# B&R Automation Studio project mappViewGettingStarted
Automation Studio 4.3.3.196; technology packages: mappView 1.3.0

## Configuration Config1

CPU PC_any, AutomationRuntime I4.33, Build 4.1.2, Vc V4.25.0

### Hardware
```
PC : PC_any v1.1.0.0 (OrderNumber=PC)
  ConfigurationID = mappViewGettingStarted_Config1
  ActivateOpcUa = 1
```

## Logical view

### Program Logical/Program (IEC)

#### Variables.var
```iecst
VAR
	MTBasicsPT1_0 : MTBasicsPT1;
	aiTankLevel : USINT;
	arrayVm : ARRAY[0..99] OF UINT;
	i : INT;
END_VAR
```

#### Main.st
```iecst
PROGRAM _INIT
	SetTemperature := 35;
END_PROGRAM

PROGRAM _CYCLIC
	(*
		Using FUNCTION block MTBasicsPT1() TO
		implement a 1st order delay element (PT1).
	*)
	MTBasicsPT1_0.Enable := 1;
	MTBasicsPT1_0.Gain := 1;
	MTBasicsPT1_0.TimeConstant := 1;
	MTBasicsPT1_0.In := INT_TO_REAL(SetTemperature);

	MTBasicsPT1_0();

	CurrentTemperature := REAL_TO_INT(MTBasicsPT1_0.Out);

	(*
		generate saw tooth signal for further usage of TM641 exercises

	*)
	aiTankLevel := aiTankLevel + 1;

	(*
		Generate values in array for LineChart
	*)
	arrayVm[0] := arrayVm[0] + 1;
	FOR i:= 1 TO 99 DO
		IF arrayVm[i] THEN
		END_IF
	END_FOR

END_PROGRAM
```

- Visualisation Logical/mappView (not shown)

Listed in the project but not available here: Logical/Global.typ, Logical/Global.var, Logical/Libraries
